{attribute 'linkalways'} 
{attribute 'no_explicit_call' := 'This FB is a CLASS and must be accessed using methods or properties'}
{attribute 'enable_dynamic_creation'}
FUNCTION_BLOCK _ETcVnOrientationMethod EXTENDS EnumDatatypeBase
VAR
	localData : ETcVnOrientationMethod;
	activeData : REFERENCE TO ETcVnOrientationMethod;
	enumBaseDatatype : _DINT(localData);
END_VAR

METHOD PRIVATE AddLocalEnumeration
VAR_INPUT
	Enumeration : T_MAXSTRING;
	Value : ETcVnOrientationMethod;
END_VAR
AddEnumeration(Enumeration, Value);
END_METHOD

PROPERTY PUBLIC Address : PVOID
GET
Address := ADR(activeData);
END_GET
END_PROPERTY

METHOD PUBLIC ClearReference
VAR_INPUT
END_VAR
activeData REF= localData;
SetBaseDatatypeReference();
END_METHOD

METHOD PUBLIC Clone : I_Datatype
VAR
    pClone : POINTER TO _ETcVnOrientationMethod;
END_VAR
pClone := __NEW(_ETcVnOrientationMethod(InitialValue := Value));
Clone := pClone^;
END_METHOD

METHOD FB_init : BOOL
VAR_INPUT
	bInitRetains : BOOL; // if TRUE, the retain variables are initialized (warm start / cold start)
	bInCopyCode : BOOL;  // if TRUE, the instance afterwards gets moved into the copy code (online change)
	InitialValue : ETcVnOrientationMethod;
END_VAR
localData := InitialValue;
AddBaseDatatype(enumBaseDatatype);
ClearReference();

AddLocalEnumeration('TCVN_OM_PCA', ETcVnOrientationMethod.TCVN_OM_PCA);
AddLocalEnumeration('TCVN_OM_FITELLIPSE', ETcVnOrientationMethod.TCVN_OM_FITELLIPSE);
AddLocalEnumeration('TCVN_OM_MOMENTS', ETcVnOrientationMethod.TCVN_OM_MOMENTS);
AddLocalEnumeration('TCVN_OM_ENCLOSINGRECT', ETcVnOrientationMethod.TCVN_OM_ENCLOSINGRECT);
END_METHOD

PROPERTY PUBLIC Identifier : T_MAXSTRING
GET
Identifier := 'ETcVnOrientationMethod';
END_GET
END_PROPERTY

METHOD IsEnumeratorValueEqual : BOOL
VAR_INPUT
	Enumerator : I_KeyValueForwardEnumerator;
END_VAR
VAR
	storedValue : ETcVnOrientationMethod;
END_VAR
IF NOT Enumerator.TryGet(storedValue) THEN
	RETURN;
END_IF

IsEnumeratorValueEqual := storedValue = activeData;
END_METHOD

METHOD PUBLIC MakeReferenceTo
VAR_INPUT
	ReferenceTarget : REFERENCE TO ETcVnOrientationMethod;
END_VAR
activeData REF= ReferenceTarget;
SetBaseDatatypeReference();
END_METHOD

METHOD PROTECTED SetBaseDatatypeReference
VAR_INPUT
END_VAR
enumBaseDatatype.MakeReferenceTo(activeData);
END_METHOD

PROPERTY PUBLIC Size : UDINT
GET
Size := SIZEOF(activeData);
END_GET
END_PROPERTY

METHOD TryMakeReferenceTo : BOOL
VAR_INPUT
	Target : I_Datatype;
END_VAR
VAR
	targetAsEnum : I_EnumDatatype;
	pTargetData : POINTER TO ETcVnOrientationMethod;
END_VAR
IF NOT Target.TryResolveAsEnumDatatype(targetAsEnum) THEN
	RETURN;
END_IF

IF targetAsEnum.Identifier <> Identifier THEN
	RETURN;
END_IF

pTargetData := Target.Address;
activeData REF= pTargetData^;
SetBaseDatatypeReference();
TryMakeReferenceTo := TRUE;
END_METHOD

PROPERTY PUBLIC Value : ETcVnOrientationMethod
GET
Value := activeData;
END_GET
SET
activeData := Value;
END_SET
END_PROPERTY

END_FUNCTION_BLOCK

(* stored: Version 1.1.0.1, ProductVersion 3.1.4024.13
   POU _ETcVnOrientationMethod: Id {0db68993-40a8-08b7-093c-5669a27ae4ce}, SpecialFunc None
   Folder Core: Id {b04d22a8-ca15-0f3f-0010-7a9c69a8f9db}
   Folder Protected: Id {a0afef9c-1251-0aed-0812-124e654ce952}
   Folder Customize: Id {aa2ba897-d92a-0235-27d0-e7f8624d6ed1}
   Folder Constructor: Id {ea42ed68-f7be-0cfd-340a-683babe80f6b}
   Folder Private: Id {586a42f0-4bc7-0255-2565-5ccaa991867e}
   Folder Protected: Id {d5d7188f-1c17-0fad-3f49-dd50ced37ff5}
   Method AddLocalEnumeration: Id {c5c5b5f3-11e3-0aaf-0398-8cc6437f121e}
   Property Address: Id {3291bcc7-91b9-0310-104b-df27fd6e2fba}
   Get Get: Id {249f6908-8f60-0abf-1c56-1ab331a6ca75}
   Method ClearReference: Id {e4c36f3c-a0c2-0356-193e-9d4f24a69334}
   Method Clone: Id {fb35618d-8b6c-09bc-00e1-90d8c75b1ab1}
   Method FB_init: Id {21322369-f54f-0af5-1094-9aec9f179013}
   Property Identifier: Id {a41bc92d-855e-0019-02ab-5cbf93d8d12f}
   Get Get: Id {d83d247d-5d0d-0305-0ece-6ae87dbf148a}
   Method IsEnumeratorValueEqual: Id {5e06bd98-3e89-0072-1e76-585aac778c16}
   Method MakeReferenceTo: Id {319985e2-bc60-0c12-3125-95d597a78ea8}
   Method SetBaseDatatypeReference: Id {2b7998cc-1049-0df3-35dc-515d82c82fab}
   Property Size: Id {9c9f7252-2dd9-055f-138c-9fb29f53908b}
   Get Get: Id {8eca2e06-e2ed-0911-369c-452f76c01d0d}
   Method TryMakeReferenceTo: Id {53887ae0-5b6e-0238-1416-00c335bdda35}
   Property Value: Id {1d78f691-ed2b-0b68-3a16-23f6c043ef68}
   Get Get: Id {02dc0329-822c-0191-3ee2-a5099cf41bde}
   Set Set: Id {7a92985a-6798-0898-1887-50c96906a82b} *)
